// TIA Portal V17 export
// export: Created 2024-08-26T21:07:22.4411771Z, ExportSetting WithDefaults, DisplayName Totally Integrated Automation Portal, DisplayVersion V17 Update 7, DisplayName TIA Portal Openness, DisplayVersion V17 Update 7, DisplayName TIA Portal Version Control Interface, DisplayVersion V17, DisplayName SINAMICS Startdrive Advanced, DisplayVersion V17 SP2, DisplayName SINAMICS Startdrive G110M, G120, G120C, G120D, G120P, G115D, DisplayVersion V17 SP2, DisplayName SINAMICS Startdrive G130, G150, S120, S150, SINAMICS MV, S210, DisplayVersion V17 SP2, DisplayName STEP 7 Professional, DisplayVersion V17 Update 7, DisplayName STEP 7 Safety, DisplayVersion V17 Update 6, DisplayName WinCC Advanced / Unified PC, DisplayVersion V17 Update 7
VAR_GLOBAL   // PLC tag table "productionMemory"
   shift1Production AT %MW300 : Int;
   shift1 AT %M350.0 : Bool;
   shift2Production AT %MW302 : Int;
   shift2 AT %M350.1 : Bool;
   shift3Production AT %MW304 : Int;
   shift3 AT %M350.2 : Bool;
   timeShift1 AT %M350.3 : Bool;
   timeShift2 AT %M350.4 : Bool;
   timeShift3 AT %M350.5 : Bool;
END_VAR
